{attribute 'qualified_only'}
{attribute 'strict'}
TYPE E_SensorBrand :
(
	Sick,
	Pilz,
	Parker,
	Bosch
);
END_TYPE

(* stored: Version 1.1.0.1, ProductVersion 3.1.4024.12
   DUT E_SensorBrand: Id {04f8bcf9-106f-475b-a61d-3ab4bf1ffd3d} *)
